FUNCTION WithinTolerance : BOOL
VAR_INPUT
	v1 : LREAL;
	v2 : LREAL;
	tolerance : LREAL;
END_VAR
(*
checks if v1 close enough to v2 within a given margin
*)

WithinTolerance := ABS(v1-v2) < tolerance;

END_FUNCTION

(* stored: Version 1.1.0.1, ProductVersion 3.1.4024.11
   POU WithinTolerance: Id {4e9ced49-a952-4cb0-b414-35672bc8309e}, SpecialFunc None *)
